Staubli VAL3: writeFloatValue.pgx

public program writeFloatValue(num handle_, num col_, num row_, num value_, bool& result_[])
  local string strCell
begin
  // write a float value into a cell
  nCommand[handle_]=coSF
  call coord2Cell(col_,row_,strCell)
  call sendCommand(handle_,"sf"+strCell+toString("0.5",value_),result_)
end
